Yaskawa INFORM job: AAA.JBI

/JOB
//NAME AAA
//POS
///NPOS 4,0,2,0,0,0
///TOOL 12
///POSTYPE PULSE
///PULSE
C00000=-35713,0,0,0,0,0
C00001=-19910,75675,-5165,-68902,-81252,69367
C00002=-35713,64940,13276,10060,-42874,-11032
C00003=-19910,75675,-5165,-68902,-81252,69367
EC00000=-29914,-208537
EC00001=-29914,-208537
//INST
///DATE 2023/10/18 18:07
///ATTR SC,RW
///GROUP1 RB1,ST1
///GROUP2 RB2
NOP
MOVJ C00000 EC00000 VJ=7.0 +MOVJ C00001
MOVJ C00002 EC00001 VJ=7.0 +MOVJ C00003
END
